// TIA Portal project "Projekt_v2" (V13)
// Vorlageprojekt für das Buch mit Zielsystem S7-1200

(* hardware
DEVICE "S7-1200-Station_1"  S7-1200 Station
   slot 0: "Baugruppenträger_0"  Rack  V1.0
   slot 1: "PLC_1"  CPU 1214C DC/DC/Rly  6ES7 214-1HG40-0XB0  V4.1
   slot 2: "DQ 16xRelay_1"  6ES7 222-1HH30-0XB0  V1.0
   slot 3: "DI 16x24VDC_1"  6ES7 221-1BH32-0XB0  V2.0
*)

// ===== PLC "PLC_1"  CPU 1214C DC/DC/Rly =====

VAR_GLOBAL   // PLC tag table "Standard-Variablentabelle"
   "Tag_2" AT %I0.0 : Bool;
   "Tag_3" AT %I0.1 : Bool;
   "Start btn" AT %I0.2 : Bool;
   "Emergency" AT %I0.4 : Bool;
   "Stop btn" AT %I0.3 : Bool;
   "Sstart" AT %I0.5 : Bool;
   "VS sorting 1" AT %ID38 : DWord;
   "VS sorting2" AT %ID34 : DWord;
   "ColorStopS" AT %I0.6 : Bool;
   "Threshold1" AT %I0.7 : Bool;
   "ResetBufor" AT %I1.0 : Bool;
   "ErrorSensor" AT %I1.1 : Bool;
   "SolveError" AT %I1.2 : Bool;
   "PallPalletAtEntry" AT %I2.0 : Bool;
   "PallPalletAtExit" AT %I2.1 : Bool;
   "PallPalletLoaded" AT %I2.2 : Bool;
   "PallBoxAtEntry" AT %I2.3 : Bool;
   "PallPusherLimit" AT %I2.4 : Bool;
   "PallPlateLimit" AT %I2.5 : Bool;
   "PallClamped" AT %I2.6 : Bool;
   "PallElevatorMoving" AT %I2.7 : Bool;
   "PallReset" AT %I1.3 : Bool;
   "Tag_1" AT %Q0.0 : Bool;
   "Start LED" AT %Q0.2 : Bool;
   "Stop LED" AT %Q0.3 : Bool;
   "ALARM" AT %Q0.4 : Bool;
   "1st Belt" AT %Q2.2 : Bool;
   "Sorter" AT %Q2.3 : Bool;
   "SorterToRight" AT %Q2.1 : Bool;
   "Arm4th" AT %Q0.7 : Bool;
   "Arm2nd" AT %Q1.0 : Bool;
   "2nd Belt" AT %Q2.4 : Bool;
   "3rd Arm" AT %Q1.1 : Bool;
   "PallPalletFeeder" AT %Q3.0 : Bool;
   "PallLoadPallet" AT %Q3.1 : Bool;
   "PallExitConveyor" AT %Q3.2 : Bool;
   "PallMoveToLimit" AT %Q3.3 : Bool;
   "PallElevatorUp" AT %Q3.4 : Bool;
   "PallElevatorDown" AT %Q3.5 : Bool;
   "PallBoxFeeder" AT %Q3.6 : Bool;
   "PallTurn" AT %Q3.7 : Bool;
   "PallPush" AT %Q4.0 : Bool;
   "PallLoadBelt" AT %Q4.1 : Bool;
   "PallClamp" AT %Q4.2 : Bool;
   "PallOpenPlate" AT %Q4.3 : Bool;
   "Priv ST" AT %M0.0 : Bool;
   "START" AT %M0.1 : Bool;
   "Tag_4" AT %M0.2 : Bool;
   "Tag_5" AT %M0.3 : Bool;
   "Tag_6" AT %M0.4 : Bool;
   "Change direction" AT %M0.5 : Bool;
   "Green Mark" AT %M1.0 : Bool;
   "BlueMark" AT %M1.1 : Bool;
   "BuforSort" AT %M8.0 : Bool;
   "FULLSORT" AT %M1.2 : Bool;
   "MetalMark" AT %M1.3 : Bool;
   "ERROR" AT %M8.2 : Bool;
   "ErrorMark" AT %M1.4 : Bool;
   "PallOpenPlateRising" AT %M3.0 : Bool;
   "PallPalletAtExitRising" AT %M3.1 : Bool;
   "PallElevatorPosition" AT %M3.2 : Bool;
   "PallBoxAtEntryRising" AT %M3.3 : Bool;
   "PallPusherLimitRising" AT %M3.4 : Bool;
   "PallPlateLimitRising" AT %M3.5 : Bool;
   "PallElevatorDownRising" AT %M3.6 : Bool;
   "PallBoxesRows" AT %MW10 : Int;
   "PallNumberBoxRows" AT %MW14 : Int;
   "PallAlturningFlag" AT %M3.7 : Bool;
   "PallPushRising" AT %M4.0 : Bool;
   "PallElevatorMovingFalling" AT %M4.1 : Bool;
   "PallPushBoxRising" AT %M4.2 : Bool;
   "PallPusherLimitFalling" AT %M4.3 : Bool;
   "PallElevatorDownRising2" AT %M4.4 : Bool;
   "SORTERisFULL" AT %M8.3 : Bool;
   "4th belt" AT %Q2.5 : Bool;
   "Arm 4th" AT %Q1.2 : Bool;
   "1st pivot" AT %Q1.3 : Bool;
   "2nd pivot" AT %Q1.4 : Bool;
   "3rd pivot" AT %Q1.5 : Bool;
   "4th pivot" AT %Q1.6 : Bool;
   "GreenTakeOFF" AT %Q0.5 : Bool;
   "BlueTakeOFF" AT %Q0.6 : Bool;
   "MetalTakeOFF" AT %Q1.7 : Bool;
   "ErrorTakeOFF" AT %Q2.0 : Bool;
END_VAR

VAR_GLOBAL CONSTANT   // PLC tag table "Standard-Variablentabelle"
   "Test" : Int := 3;
END_VAR

// folder: System blocks/Program resources

DATA_BLOCK "IEC_Timer_0_DB"   // DB1
{ S7_Optimized_Access := 'FALSE' }
AUTHOR : Simatic
FAMILY : IEC
NAME : IEC_TMR
VERSION : 1.0
// stored: InstanceOfName ?
"?"
BEGIN
END_DATA_BLOCK

DATA_BLOCK "IEC_Timer_0_DB_1"   // DB2
{ S7_Optimized_Access := 'FALSE' }
AUTHOR : Simatic
FAMILY : IEC
NAME : IEC_TMR
VERSION : 1.0
// stored: InstanceOfName ?
"?"
BEGIN
END_DATA_BLOCK

DATA_BLOCK "IEC_Timer_0_DB_2"   // DB3
{ S7_Optimized_Access := 'FALSE' }
AUTHOR : Simatic
FAMILY : IEC
NAME : IEC_TMR
VERSION : 1.0
// stored: InstanceOfName ?
"?"
BEGIN
END_DATA_BLOCK

DATA_BLOCK "IEC_Timer_0_DB_3"   // DB4
{ S7_Optimized_Access := 'FALSE' }
AUTHOR : Simatic
FAMILY : IEC
NAME : IEC_TMR
VERSION : 1.0
// stored: InstanceOfName ?
"?"
BEGIN
END_DATA_BLOCK

DATA_BLOCK "IEC_Timer_0_DB_4"   // DB5
{ S7_Optimized_Access := 'FALSE' }
AUTHOR : Simatic
FAMILY : IEC
NAME : IEC_TMR
VERSION : 1.0
// stored: InstanceOfName ?
"?"
BEGIN
END_DATA_BLOCK

DATA_BLOCK "IEC_Timer_0_DB_5"   // DB6
{ S7_Optimized_Access := 'FALSE' }
AUTHOR : Simatic
FAMILY : IEC
NAME : IEC_TMR
VERSION : 1.0
// stored: InstanceOfName ?
"?"
BEGIN
END_DATA_BLOCK

DATA_BLOCK "IEC_Timer_0_DB_6"   // DB7
{ S7_Optimized_Access := 'FALSE' }
AUTHOR : Simatic
FAMILY : IEC
NAME : IEC_TMR
VERSION : 1.0
// stored: InstanceOfName ?
"?"
BEGIN
END_DATA_BLOCK

DATA_BLOCK "Layer_Counter"   // DB8
{ S7_Optimized_Access := 'FALSE' }
AUTHOR : Simatic
FAMILY : IEC
NAME : CNTR
VERSION : 1.0
// stored: InstanceOfName ?
"?"
BEGIN
END_DATA_BLOCK

DATA_BLOCK "Off_Delay_Timer"   // DB10
{ S7_Optimized_Access := 'FALSE' }
AUTHOR : Simatic
FAMILY : IEC
NAME : IEC_TMR
VERSION : 1.0
// stored: InstanceOfName ?
"?"
BEGIN
END_DATA_BLOCK

DATA_BLOCK "Boxes_In_Row"   // DB11
{ S7_Optimized_Access := 'FALSE' }
AUTHOR : Simatic
FAMILY : IEC
NAME : CNTR
VERSION : 1.0
// stored: InstanceOfName ?
"?"
BEGIN
END_DATA_BLOCK

DATA_BLOCK "Number_of_Row"   // DB12
{ S7_Optimized_Access := 'FALSE' }
AUTHOR : Simatic
FAMILY : IEC
NAME : CNTR
VERSION : 1.0
// stored: InstanceOfName ?
"?"
BEGIN
END_DATA_BLOCK

DATA_BLOCK "Pall_Push_Timer"   // DB14
{ S7_Optimized_Access := 'FALSE' }
AUTHOR : Simatic
FAMILY : IEC
NAME : IEC_TMR
VERSION : 1.0
// stored: InstanceOfName ?
"?"
BEGIN
END_DATA_BLOCK

DATA_BLOCK "Pall_Open_Plate_Timer"   // DB15
{ S7_Optimized_Access := 'FALSE' }
AUTHOR : Simatic
FAMILY : IEC
NAME : IEC_TMR
VERSION : 1.0
// stored: InstanceOfName ?
"?"
BEGIN
END_DATA_BLOCK

// folder: (top level)

FUNCTION "Program" : Void   // FC1, LAD
{ S7_Optimized_Access := 'FALSE' }
VERSION : 0.1
   VAR_TEMP   // added for the SCL form of the ladder/FBD networks
      _w1 : Bool;
   END_VAR
BEGIN

REGION Network 1
   // Status: Start
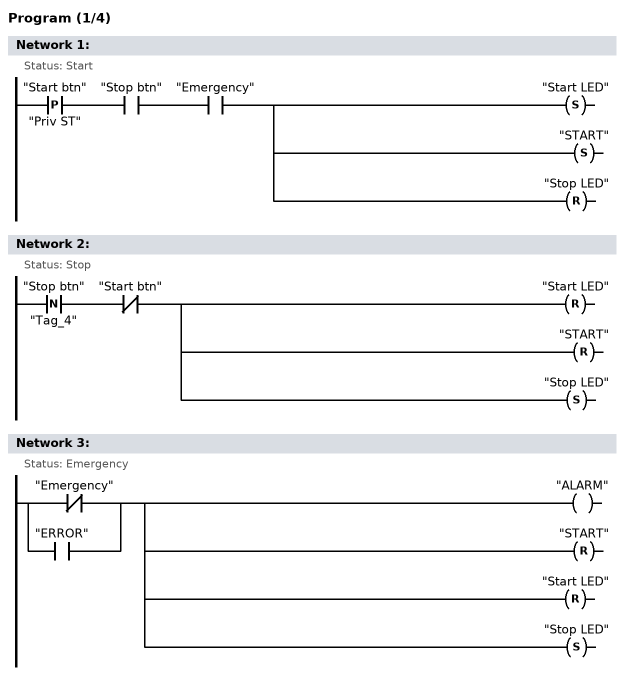
   RUNG wire#powerrail
      P_Contact(operand := "Start btn", bit := "Priv ST")
      Contact( "Stop btn" )
      Contact( "Emergency" )
      wire#w1
      S_Coil( "Start LED" )
   END_RUNG
   RUNG wire#w1
      S_Coil( "START" )
   END_RUNG
   RUNG wire#w1
      R_Coil( "Stop LED" )
   END_RUNG
   // the same network as SCL:
   #_w1 := "Start btn" AND NOT "Priv ST";   // rising edge of "Start btn"
   "Priv ST" := "Start btn";
   IF #_w1 AND "Stop btn" AND "Emergency" THEN
       "Start LED" := TRUE;
       "START" := TRUE;
       "Stop LED" := FALSE;
   END_IF;
END_REGION

REGION Network 2
   // Status: Stop
   RUNG wire#powerrail
      N_Contact(operand := "Stop btn", bit := "Tag_4")
      I_Contact( "Start btn" )
      wire#w1
      R_Coil( "Start LED" )
   END_RUNG
   RUNG wire#w1
      R_Coil( "START" )
   END_RUNG
   RUNG wire#w1
      S_Coil( "Stop LED" )
   END_RUNG
   // the same network as SCL:
   #_w1 := NOT "Stop btn" AND "Tag_4";   // falling edge of "Stop btn"
   "Tag_4" := "Stop btn";
   IF #_w1 AND NOT "Start btn" THEN
       "Start LED" := FALSE;
       "START" := FALSE;
       "Stop LED" := TRUE;
   END_IF;
END_REGION

REGION Network 3
   // Status: Emergency
   RUNG wire#powerrail
      I_Contact( "Emergency" )
      wire#w1
      Coil( "ALARM" )
   END_RUNG
   RUNG wire#powerrail
      Contact( "ERROR" )
   END_RUNG wire#w1
   RUNG wire#w1
      R_Coil( "START" )
   END_RUNG
   RUNG wire#w1
      R_Coil( "Start LED" )
   END_RUNG
   RUNG wire#w1
      S_Coil( "Stop LED" )
   END_RUNG
   // the same network as SCL:
   "ALARM" := NOT "Emergency" OR "ERROR";
   IF "ALARM" THEN
       "START" := FALSE;
       "Start LED" := FALSE;
       "Stop LED" := TRUE;
   END_IF;
END_REGION

REGION Network 4
   // 1st settings
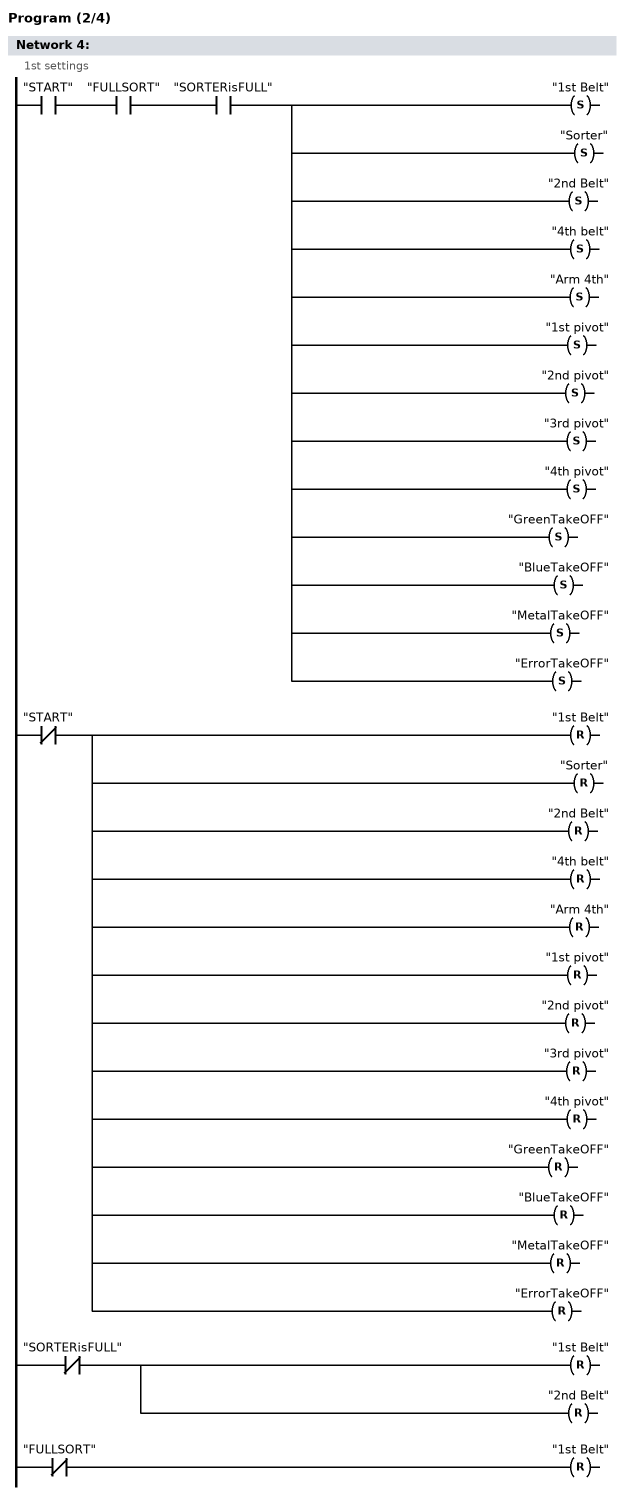
   RUNG wire#powerrail
      Contact( "START" )
      Contact( "FULLSORT" )
      Contact( "SORTERisFULL" )
      wire#w1
      S_Coil( "1st Belt" )
   END_RUNG
   RUNG wire#w1
      S_Coil( "Sorter" )
   END_RUNG
   RUNG wire#w1
      S_Coil( "2nd Belt" )
   END_RUNG
   RUNG wire#w1
      S_Coil( "4th belt" )
   END_RUNG
   RUNG wire#w1
      S_Coil( "Arm 4th" )
   END_RUNG
   RUNG wire#w1
      S_Coil( "1st pivot" )
   END_RUNG
   RUNG wire#w1
      S_Coil( "2nd pivot" )
   END_RUNG
   RUNG wire#w1
      S_Coil( "3rd pivot" )
   END_RUNG
   RUNG wire#w1
      S_Coil( "4th pivot" )
   END_RUNG
   RUNG wire#w1
      S_Coil( "GreenTakeOFF" )
   END_RUNG
   RUNG wire#w1
      S_Coil( "BlueTakeOFF" )
   END_RUNG
   RUNG wire#w1
      S_Coil( "MetalTakeOFF" )
   END_RUNG
   RUNG wire#w1
      S_Coil( "ErrorTakeOFF" )
   END_RUNG
   RUNG wire#powerrail
      I_Contact( "START" )
      wire#w2
      R_Coil( "1st Belt" )
   END_RUNG
   RUNG wire#w2
      R_Coil( "Sorter" )
   END_RUNG
   RUNG wire#w2
      R_Coil( "2nd Belt" )
   END_RUNG
   RUNG wire#w2
      R_Coil( "4th belt" )
   END_RUNG
   RUNG wire#w2
      R_Coil( "Arm 4th" )
   END_RUNG
   RUNG wire#w2
      R_Coil( "1st pivot" )
   END_RUNG
   RUNG wire#w2
      R_Coil( "2nd pivot" )
   END_RUNG
   RUNG wire#w2
      R_Coil( "3rd pivot" )
   END_RUNG
   RUNG wire#w2
      R_Coil( "4th pivot" )
   END_RUNG
   RUNG wire#w2
      R_Coil( "GreenTakeOFF" )
   END_RUNG
   RUNG wire#w2
      R_Coil( "BlueTakeOFF" )
   END_RUNG
   RUNG wire#w2
      R_Coil( "MetalTakeOFF" )
   END_RUNG
   RUNG wire#w2
      R_Coil( "ErrorTakeOFF" )
   END_RUNG
   RUNG wire#powerrail
      I_Contact( "SORTERisFULL" )
      wire#w3
      R_Coil( "1st Belt" )
   END_RUNG
   RUNG wire#w3
      R_Coil( "2nd Belt" )
   END_RUNG
   RUNG wire#powerrail
      I_Contact( "FULLSORT" )
      R_Coil( "1st Belt" )
   END_RUNG
   // the same network as SCL:
   IF "START" AND "FULLSORT" AND "SORTERisFULL" THEN
       "1st Belt" := TRUE;
       "Sorter" := TRUE;
       "2nd Belt" := TRUE;
       "4th belt" := TRUE;
       "Arm 4th" := TRUE;
       "1st pivot" := TRUE;
       "2nd pivot" := TRUE;
       "3rd pivot" := TRUE;
       "4th pivot" := TRUE;
       "GreenTakeOFF" := TRUE;
       "BlueTakeOFF" := TRUE;
       "MetalTakeOFF" := TRUE;
       "ErrorTakeOFF" := TRUE;
   END_IF;
   IF NOT "START" THEN
       "1st Belt" := FALSE;
       "Sorter" := FALSE;
       "2nd Belt" := FALSE;
       "4th belt" := FALSE;
       "Arm 4th" := FALSE;
       "1st pivot" := FALSE;
       "2nd pivot" := FALSE;
       "3rd pivot" := FALSE;
       "4th pivot" := FALSE;
       "GreenTakeOFF" := FALSE;
       "BlueTakeOFF" := FALSE;
       "MetalTakeOFF" := FALSE;
       "ErrorTakeOFF" := FALSE;
   END_IF;
   IF NOT "SORTERisFULL" THEN
       "1st Belt" := FALSE;
       "2nd Belt" := FALSE;
   END_IF;
   IF NOT "FULLSORT" THEN "1st Belt" := FALSE; END_IF;
END_REGION

REGION Network 5
   // 1st sorting boxes vs color things
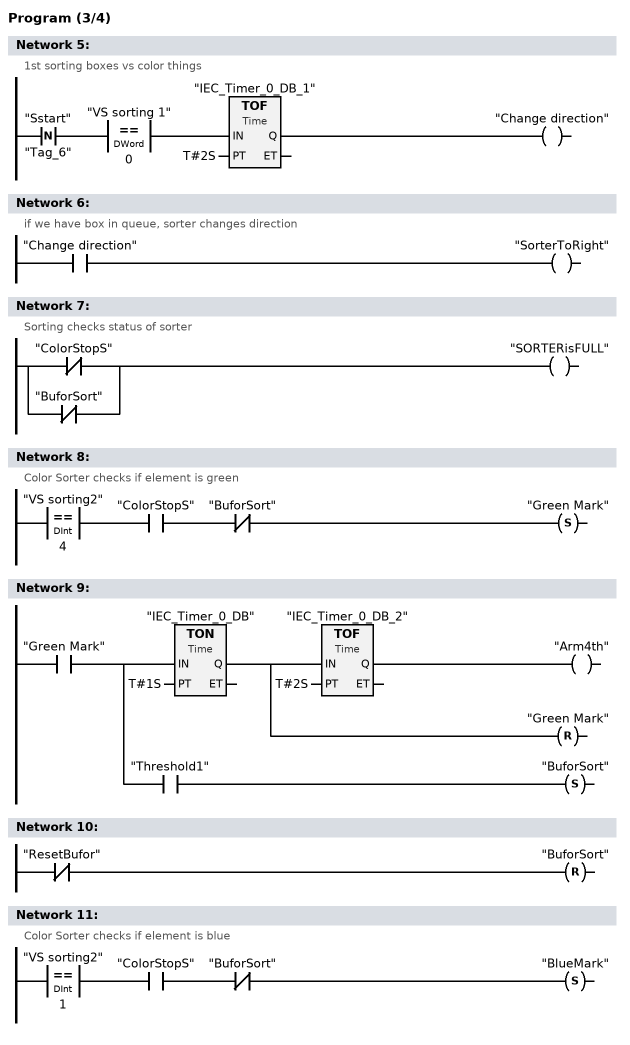
   #_w1 := NOT "Sstart" AND "Tag_6";   // falling edge of "Sstart"
   "Tag_6" := "Sstart";
   "IEC_Timer_0_DB_1".TOF(IN := #_w1 AND ("VS sorting 1" = 0), PT := T#2S);
   "Change direction" := "IEC_Timer_0_DB_1".Q;
END_REGION

REGION Network 6
   // if we have box in queue, sorter changes direction
   RUNG wire#powerrail
      Contact( "Change direction" )
      Coil( "SorterToRight" )
   END_RUNG
   // the same network as SCL:
   "SorterToRight" := "Change direction";
END_REGION

REGION Network 7
   // Sorting checks status of sorter
   RUNG wire#powerrail
      I_Contact( "ColorStopS" )
      wire#w1
      Coil( "SORTERisFULL" )
   END_RUNG
   RUNG wire#powerrail
      I_Contact( "BuforSort" )
   END_RUNG wire#w1
   // the same network as SCL:
   "SORTERisFULL" := NOT "ColorStopS" OR NOT "BuforSort";
END_REGION

REGION Network 8
   // Color Sorter checks if element is green
   RUNG wire#powerrail
      { S7_Templates := "SrcType := DInt" } EQ_Contact(in1 := "VS sorting2", in2 := 4)
      Contact( "ColorStopS" )
      I_Contact( "BuforSort" )
      S_Coil( "Green Mark" )
   END_RUNG
   // the same network as SCL:
   IF ("VS sorting2" = 4) AND "ColorStopS" AND NOT "BuforSort" THEN "Green Mark" := TRUE; END_IF;
END_REGION

REGION Network 9
   "IEC_Timer_0_DB".TON(IN := "Green Mark", PT := T#1S);
   "IEC_Timer_0_DB_2".TOF(IN := "IEC_Timer_0_DB".Q, PT := T#2S);
   "Arm4th" := "IEC_Timer_0_DB_2".Q;
   #_w1 := "Green Mark";
   IF "IEC_Timer_0_DB".Q THEN "Green Mark" := FALSE; END_IF;
   IF #_w1 AND "Threshold1" THEN "BuforSort" := TRUE; END_IF;
END_REGION

REGION Network 10
   RUNG wire#powerrail
      I_Contact( "ResetBufor" )
      R_Coil( "BuforSort" )
   END_RUNG
   // the same network as SCL:
   IF NOT "ResetBufor" THEN "BuforSort" := FALSE; END_IF;
END_REGION

REGION Network 11
   // Color Sorter checks if element is blue
   RUNG wire#powerrail
      { S7_Templates := "SrcType := DInt" } EQ_Contact(in1 := "VS sorting2", in2 := 1)
      Contact( "ColorStopS" )
      I_Contact( "BuforSort" )
      S_Coil( "BlueMark" )
   END_RUNG
   // the same network as SCL:
   IF ("VS sorting2" = 1) AND "ColorStopS" AND NOT "BuforSort" THEN "BlueMark" := TRUE; END_IF;
END_REGION

REGION Network 12
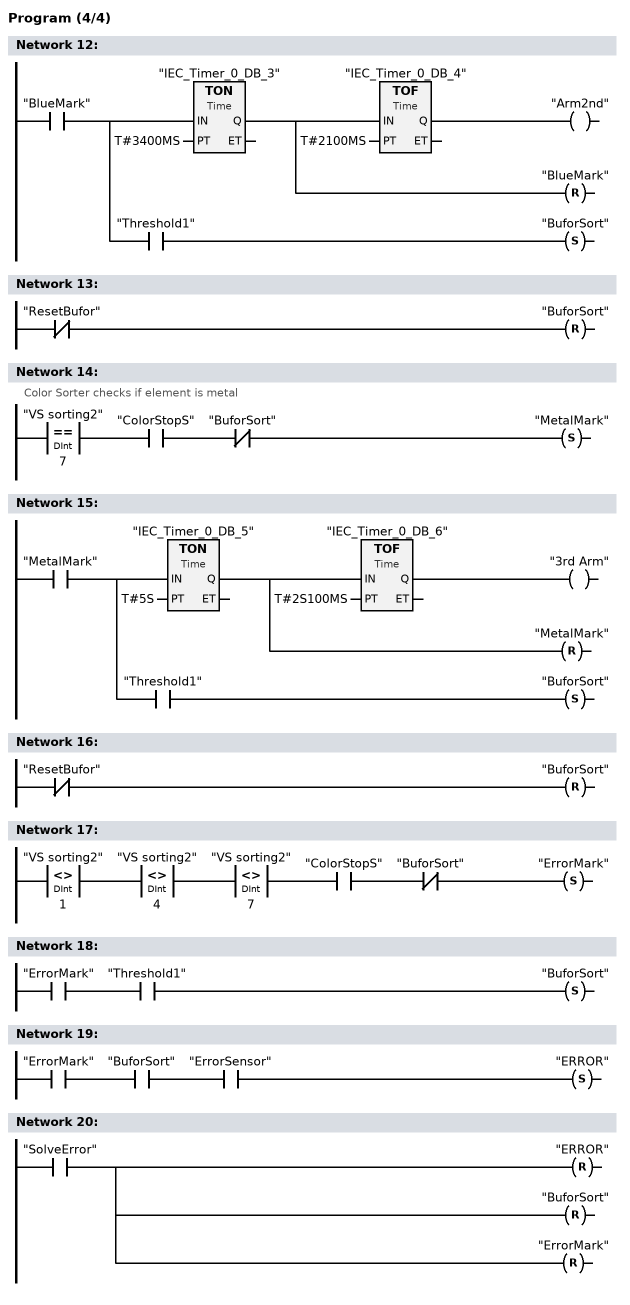
   "IEC_Timer_0_DB_3".TON(IN := "BlueMark", PT := T#3400MS);
   "IEC_Timer_0_DB_4".TOF(IN := "IEC_Timer_0_DB_3".Q, PT := T#2100MS);
   "Arm2nd" := "IEC_Timer_0_DB_4".Q;
   #_w1 := "BlueMark";
   IF "IEC_Timer_0_DB_3".Q THEN "BlueMark" := FALSE; END_IF;
   IF #_w1 AND "Threshold1" THEN "BuforSort" := TRUE; END_IF;
END_REGION

REGION Network 13
   RUNG wire#powerrail
      I_Contact( "ResetBufor" )
      R_Coil( "BuforSort" )
   END_RUNG
   // the same network as SCL:
   IF NOT "ResetBufor" THEN "BuforSort" := FALSE; END_IF;
END_REGION

REGION Network 14
   // Color Sorter checks if element is metal
   RUNG wire#powerrail
      { S7_Templates := "SrcType := DInt" } EQ_Contact(in1 := "VS sorting2", in2 := 7)
      Contact( "ColorStopS" )
      I_Contact( "BuforSort" )
      S_Coil( "MetalMark" )
   END_RUNG
   // the same network as SCL:
   IF ("VS sorting2" = 7) AND "ColorStopS" AND NOT "BuforSort" THEN "MetalMark" := TRUE; END_IF;
END_REGION

REGION Network 15
   "IEC_Timer_0_DB_5".TON(IN := "MetalMark", PT := T#5S);
   "IEC_Timer_0_DB_6".TOF(IN := "IEC_Timer_0_DB_5".Q, PT := T#2S100MS);
   "3rd Arm" := "IEC_Timer_0_DB_6".Q;
   #_w1 := "MetalMark";
   IF "IEC_Timer_0_DB_5".Q THEN "MetalMark" := FALSE; END_IF;
   IF #_w1 AND "Threshold1" THEN "BuforSort" := TRUE; END_IF;
END_REGION

REGION Network 16
   RUNG wire#powerrail
      I_Contact( "ResetBufor" )
      R_Coil( "BuforSort" )
   END_RUNG
   // the same network as SCL:
   IF NOT "ResetBufor" THEN "BuforSort" := FALSE; END_IF;
END_REGION

REGION Network 17
   RUNG wire#powerrail
      { S7_Templates := "SrcType := DInt" } NE_Contact(in1 := "VS sorting2", in2 := 1)
      { S7_Templates := "SrcType := DInt" } NE_Contact(in1 := "VS sorting2", in2 := 4)
      { S7_Templates := "SrcType := DInt" } NE_Contact(in1 := "VS sorting2", in2 := 7)
      Contact( "ColorStopS" )
      I_Contact( "BuforSort" )
      S_Coil( "ErrorMark" )
   END_RUNG
   // the same network as SCL:
   IF ("VS sorting2" <> 1) AND ("VS sorting2" <> 4) AND ("VS sorting2" <> 7) AND "ColorStopS" AND NOT "BuforSort" THEN
       "ErrorMark" := TRUE;
   END_IF;
END_REGION

REGION Network 18
   RUNG wire#powerrail
      Contact( "ErrorMark" )
      Contact( "Threshold1" )
      S_Coil( "BuforSort" )
   END_RUNG
   // the same network as SCL:
   IF "ErrorMark" AND "Threshold1" THEN "BuforSort" := TRUE; END_IF;
END_REGION

REGION Network 19
   RUNG wire#powerrail
      Contact( "ErrorMark" )
      Contact( "BuforSort" )
      Contact( "ErrorSensor" )
      S_Coil( "ERROR" )
   END_RUNG
   // the same network as SCL:
   IF "ErrorMark" AND "BuforSort" AND "ErrorSensor" THEN "ERROR" := TRUE; END_IF;
END_REGION

REGION Network 20
   RUNG wire#powerrail
      Contact( "SolveError" )
      wire#w1
      R_Coil( "ERROR" )
   END_RUNG
   RUNG wire#w1
      R_Coil( "BuforSort" )
   END_RUNG
   RUNG wire#w1
      R_Coil( "ErrorMark" )
   END_RUNG
   // the same network as SCL:
   IF "SolveError" THEN
       "ERROR" := FALSE;
       "BuforSort" := FALSE;
       "ErrorMark" := FALSE;
   END_IF;
END_REGION
END_FUNCTION

FUNCTION "Palletizer" : Void   // FC2, LAD
{ S7_Optimized_Access := 'FALSE' }
VERSION : 0.1
   VAR_TEMP   // added for the SCL form of the ladder/FBD networks
      _w1 : Bool;
      _w2 : Bool;
      _w3 : Bool;
      _w4 : Bool;
      _w5 : Bool;
      _w6 : Bool;
      _w7 : Bool;
      _w8 : Bool;
      _w9 : Bool;
      _w10 : Bool;
      _w11 : Bool;
   END_VAR
BEGIN

REGION Network 1: Loading / Unloading Pallets
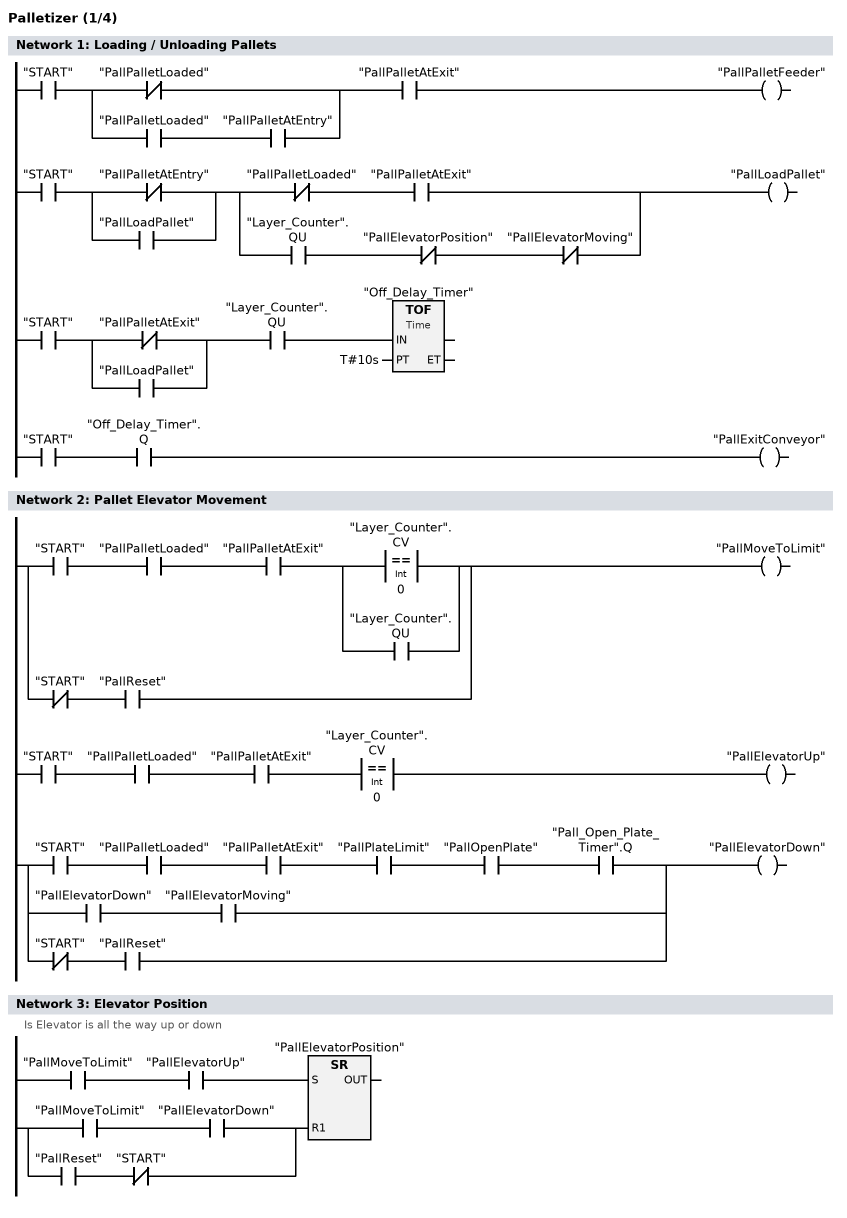
   "PallPalletFeeder" := "START" AND (NOT "PallPalletLoaded" OR ("PallPalletLoaded" AND "PallPalletAtEntry")) AND "PallPalletAtExit";
   "PallLoadPallet" := "START" AND (NOT "PallPalletAtEntry" OR "PallLoadPallet") AND ((NOT "PallPalletLoaded" AND "PallPalletAtExit") OR ("Layer_Counter".QU AND NOT "PallElevatorPosition" AND NOT "PallElevatorMoving"));
   "Off_Delay_Timer".TOF(IN := "START" AND (NOT "PallPalletAtExit" OR "PallLoadPallet") AND "Layer_Counter".QU,
                         PT := T#10s);
   "PallExitConveyor" := "START" AND "Off_Delay_Timer".Q;
END_REGION

REGION Network 2: Pallet Elevator Movement
   RUNG wire#powerrail
      Contact( "START" )
      Contact( "PallPalletLoaded" )
      Contact( "PallPalletAtExit" )
      wire#w1
      { S7_Templates := "SrcType := Int" } EQ_Contact(in1 := "Layer_Counter".CV, in2 := 0)
      wire#w2
      Coil( "PallMoveToLimit" )
   END_RUNG
   RUNG wire#w1
      Contact( "Layer_Counter".QU )
   END_RUNG wire#w2
   RUNG wire#powerrail
      I_Contact( "START" )
      Contact( "PallReset" )
   END_RUNG wire#w2
   RUNG wire#powerrail
      Contact( "START" )
      Contact( "PallPalletLoaded" )
      Contact( "PallPalletAtExit" )
      { S7_Templates := "SrcType := Int" } EQ_Contact(in1 := "Layer_Counter".CV, in2 := 0)
      Coil( "PallElevatorUp" )
   END_RUNG
   RUNG wire#powerrail
      Contact( "START" )
      Contact( "PallPalletLoaded" )
      Contact( "PallPalletAtExit" )
      Contact( "PallPlateLimit" )
      Contact( "PallOpenPlate" )
      Contact( "Pall_Open_Plate_Timer".Q )
      wire#w3
      Coil( "PallElevatorDown" )
   END_RUNG
   RUNG wire#powerrail
      Contact( "PallElevatorDown" )
      Contact( "PallElevatorMoving" )
   END_RUNG wire#w3
   RUNG wire#powerrail
      I_Contact( "START" )
      Contact( "PallReset" )
   END_RUNG wire#w3
   // the same network as SCL:
   "PallMoveToLimit" := ("START" AND "PallPalletLoaded" AND "PallPalletAtExit" AND (("Layer_Counter".CV = 0) OR "Layer_Counter".QU)) OR (NOT "START" AND "PallReset");
   "PallElevatorUp" := "START" AND "PallPalletLoaded" AND "PallPalletAtExit" AND ("Layer_Counter".CV = 0);
   "PallElevatorDown" := ("START" AND "PallPalletLoaded" AND "PallPalletAtExit" AND "PallPlateLimit" AND "PallOpenPlate" AND "Pall_Open_Plate_Timer".Q) OR ("PallElevatorDown" AND "PallElevatorMoving") OR (NOT "START" AND "PallReset");
END_REGION

REGION Network 3: Elevator Position
   // Is Elevator is all the way up or down
   RUNG wire#powerrail
      Contact( "PallMoveToLimit" )
      Contact( "PallElevatorUp" )
      S_SR(operand := "PallElevatorPosition", r1 := wire#w1)
   END_RUNG
   RUNG wire#powerrail
      Contact( "PallMoveToLimit" )
      Contact( "PallElevatorDown" )
   END_RUNG wire#w1
   RUNG wire#powerrail
      Contact( "PallReset" )
      I_Contact( "START" )
   END_RUNG wire#w1
   // the same network as SCL:
   IF "PallMoveToLimit" AND "PallElevatorUp" THEN
       "PallElevatorPosition" := TRUE;   // SR flip-flop
   END_IF;
   IF ("PallMoveToLimit" AND "PallElevatorDown") OR ("PallReset" AND NOT "START") THEN
       "PallElevatorPosition" := FALSE;
   END_IF;
END_REGION

REGION Network 4: Number of Layers on the Pallet
   // Couter tracks how many layers are on pallet
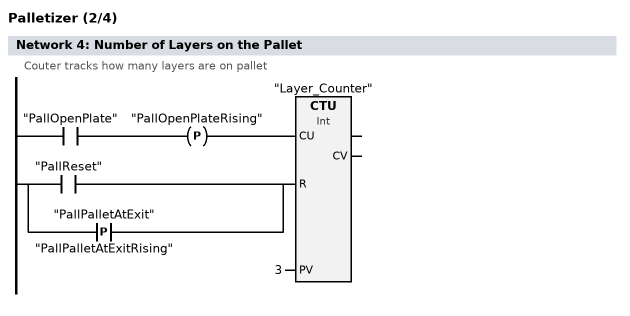
   #_w1 := "PallOpenPlate" AND NOT "PallOpenPlateRising";   // rising edge
   "PallOpenPlateRising" := "PallOpenPlate";
   #_w2 := "PallPalletAtExit" AND NOT "PallPalletAtExitRising";   // rising edge of "PallPalletAtExit"
   "PallPalletAtExitRising" := "PallPalletAtExit";
   "Layer_Counter".CTU(CU := #_w1, R := "PallReset" OR #_w2, PV := 3);
END_REGION

REGION Network 5: Boxes on Layers
   // 6 boxes on layer. Each Layer is alturnating
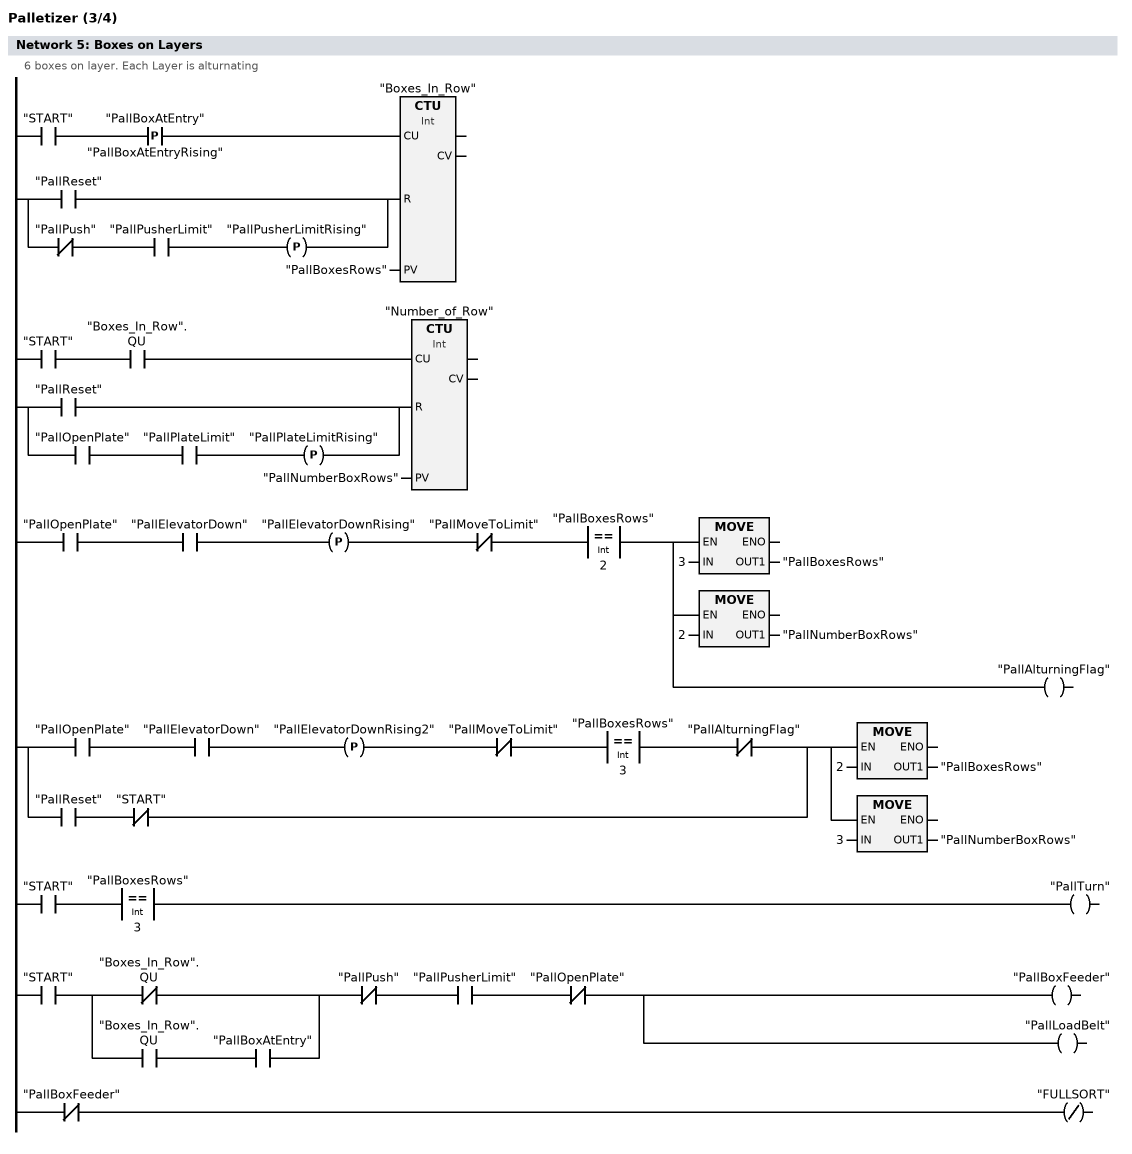
   #_w1 := "START" AND "PallBoxAtEntry" AND NOT "PallBoxAtEntryRising";   // rising edge of "PallBoxAtEntry"
   "PallBoxAtEntryRising" := "PallBoxAtEntry";
   #_w2 := NOT "PallPush" AND "PallPusherLimit";
   #_w3 := #_w2 AND NOT "PallPusherLimitRising";   // rising edge
   "PallPusherLimitRising" := #_w2;
   "Boxes_In_Row".CTU(CU := #_w1, R := "PallReset" OR #_w3, PV := "PallBoxesRows");
   #_w4 := "PallOpenPlate" AND "PallPlateLimit";
   #_w5 := #_w4 AND NOT "PallPlateLimitRising";   // rising edge
   "PallPlateLimitRising" := #_w4;
   "Number_of_Row".CTU(CU := "START" AND "Boxes_In_Row".QU, R := "PallReset" OR #_w5, PV := "PallNumberBoxRows");
   #_w6 := "PallOpenPlate" AND "PallElevatorDown";
   #_w7 := #_w6 AND NOT "PallElevatorDownRising";   // rising edge
   "PallElevatorDownRising" := #_w6;
   #_w8 := #_w7 AND NOT "PallMoveToLimit" AND ("PallBoxesRows" = 2);
   IF #_w8 THEN
       "PallBoxesRows" := 3;
       "PallNumberBoxRows" := 2;
   END_IF;
   "PallAlturningFlag" := #_w8;
   #_w9 := "PallOpenPlate" AND "PallElevatorDown";
   #_w10 := #_w9 AND NOT "PallElevatorDownRising2";   // rising edge
   "PallElevatorDownRising2" := #_w9;
   #_w11 := (#_w10 AND NOT "PallMoveToLimit" AND ("PallBoxesRows" = 3) AND NOT "PallAlturningFlag") OR ("PallReset" AND NOT "START");
   IF #_w11 THEN
       "PallBoxesRows" := 2;
       "PallNumberBoxRows" := 3;
   END_IF;
   "PallTurn" := "START" AND ("PallBoxesRows" = 3);
   "PallBoxFeeder" := "START" AND (NOT "Boxes_In_Row".QU OR ("Boxes_In_Row".QU AND "PallBoxAtEntry")) AND NOT "PallPush" AND "PallPusherLimit" AND NOT "PallOpenPlate";
   "PallLoadBelt" := "PallBoxFeeder";
   "FULLSORT" := NOT (NOT "PallBoxFeeder");
END_REGION

REGION Network 6: Box Pusher
   // The pusher will push the boxes in the row onto the plate.
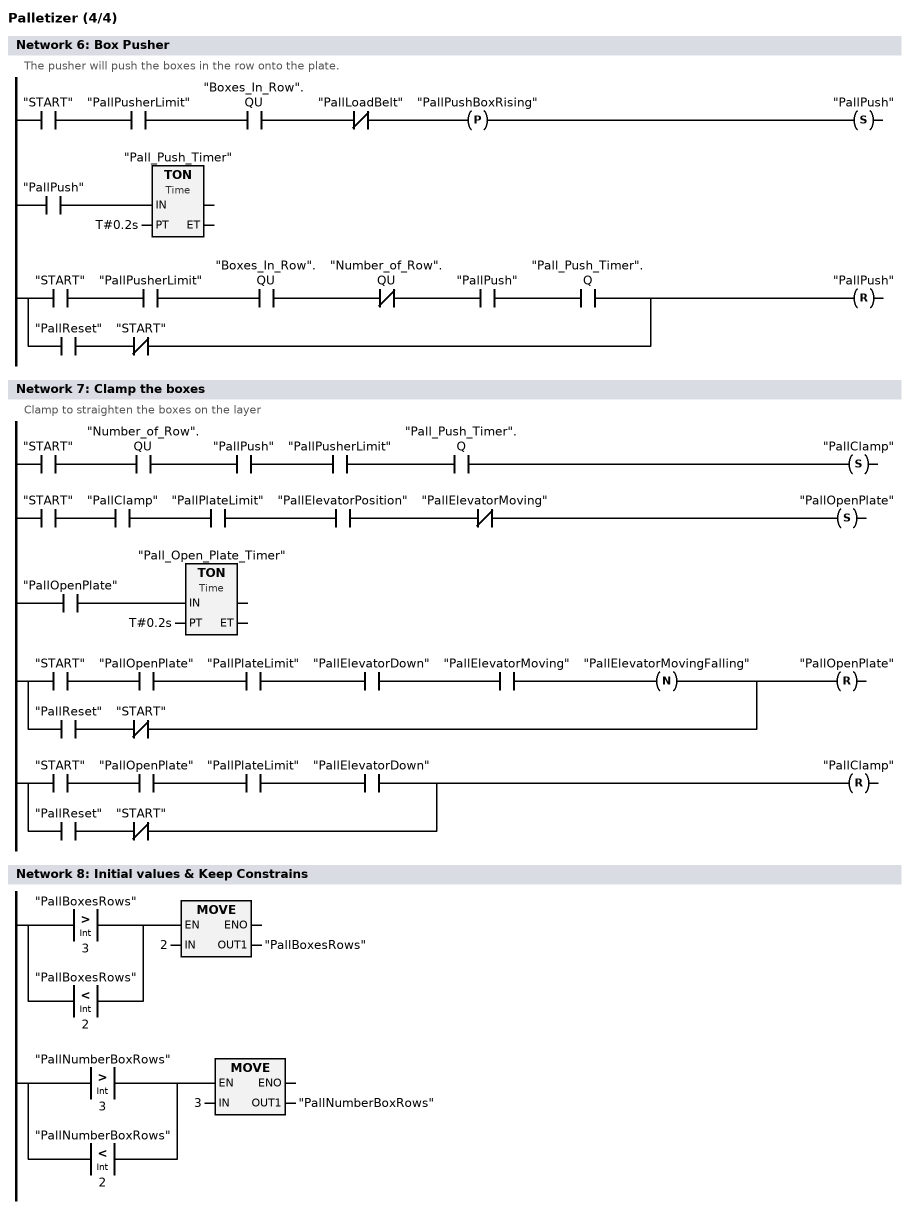
   #_w1 := "START" AND "PallPusherLimit" AND "Boxes_In_Row".QU AND NOT "PallLoadBelt";
   #_w2 := #_w1 AND NOT "PallPushBoxRising";   // rising edge
   "PallPushBoxRising" := #_w1;
   IF #_w2 THEN "PallPush" := TRUE; END_IF;
   "Pall_Push_Timer".TON(IN := "PallPush", PT := T#0.2s);
   IF ("START" AND "PallPusherLimit" AND "Boxes_In_Row".QU AND NOT "Number_of_Row".QU AND "PallPush" AND "Pall_Push_Timer".Q) OR ("PallReset" AND NOT "START") THEN
       "PallPush" := FALSE;
   END_IF;
END_REGION

REGION Network 7: Clamp the boxes
   // Clamp to straighten the boxes on the layer
   IF "START" AND "Number_of_Row".QU AND "PallPush" AND "PallPusherLimit" AND "Pall_Push_Timer".Q THEN
       "PallClamp" := TRUE;
   END_IF;
   IF "START" AND "PallClamp" AND "PallPlateLimit" AND "PallElevatorPosition" AND NOT "PallElevatorMoving" THEN
       "PallOpenPlate" := TRUE;
   END_IF;
   "Pall_Open_Plate_Timer".TON(IN := "PallOpenPlate", PT := T#0.2s);
   #_w1 := "START" AND "PallOpenPlate" AND "PallPlateLimit" AND "PallElevatorDown" AND "PallElevatorMoving";
   #_w2 := NOT #_w1 AND "PallElevatorMovingFalling";   // falling edge
   "PallElevatorMovingFalling" := #_w1;
   IF #_w2 OR ("PallReset" AND NOT "START") THEN "PallOpenPlate" := FALSE; END_IF;
   IF ("START" AND "PallOpenPlate" AND "PallPlateLimit" AND "PallElevatorDown") OR ("PallReset" AND NOT "START") THEN
       "PallClamp" := FALSE;
   END_IF;
END_REGION

REGION Network 8: Initial values & Keep Constrains
   RUNG wire#powerrail
      { S7_Templates := "SrcType := Int" } GT_Contact(in1 := "PallBoxesRows", in2 := 3)
      wire#w1
      Move(in := 2, out1 => "PallBoxesRows")
   END_RUNG
   RUNG wire#powerrail
      { S7_Templates := "SrcType := Int" } LT_Contact(in1 := "PallBoxesRows", in2 := 2)
   END_RUNG wire#w1
   RUNG wire#powerrail
      { S7_Templates := "SrcType := Int" } GT_Contact(in1 := "PallNumberBoxRows", in2 := 3)
      wire#w2
      Move(in := 3, out1 => "PallNumberBoxRows")
   END_RUNG
   RUNG wire#powerrail
      { S7_Templates := "SrcType := Int" } LT_Contact(in1 := "PallNumberBoxRows", in2 := 2)
   END_RUNG wire#w2
   // the same network as SCL:
   IF ("PallBoxesRows" > 3) OR ("PallBoxesRows" < 2) THEN "PallBoxesRows" := 2; END_IF;
   IF ("PallNumberBoxRows" > 3) OR ("PallNumberBoxRows" < 2) THEN "PallNumberBoxRows" := 3; END_IF;
END_REGION
END_FUNCTION

FUNCTION "MHJ-PLC-Lab-Function-S71200" : Void   // FC9000, SCL
{ S7_Optimized_Access := 'FALSE' }
VERSION : 0.1
BEGIN

   #Value:=PEEK(area := 16#82,
        dbNumber := 0,
        byteOffset := 511);
   #Value := #Value + 1;

   POKE(area := 16#82,
        dbNumber := 0,
        byteOffset := 511,
        value := #Value);

   POKE(area:=16#81,
        dbNumber:=0,
        byteOffset:=1016,
        value:=#Value_01_DW);
   POKE(area := 16#81,
        dbNumber := 0,
        byteOffset := 1020,
        value := #Value_02_DW);

   POKE(area := 16#81,
        dbNumber := 0,
        byteOffset := 511,
        value := B#16#00);

   FOR #forVal := 0 TO 120 DO
       FOR #forVal_2:=0 TO 10 DO
           #rdTimeReturn:=RD_SYS_T(#outputTime);
           #rdTimeReturn := WR_SYS_T(#outputTime);
           #rdTimeReturn := RD_SYS_T(#outputTime);
           #rdTimeReturn := WR_SYS_T(#outputTime);
       END_FOR;
       #SyncVal:= PEEK(area := 16#81,
                      dbNumber := 0,
                      byteOffset := 511);
       IF #SyncVal = #CompVal THEN
          GOTO M_1;
       END_IF;
   END_FOR;
   RETURN;

   M_1:
   POKE(area := 16#81,
        dbNumber := 0,
        byteOffset := 511,
        value := B#16#0);
END_FUNCTION

ORGANIZATION_BLOCK "Main"   // OB1, FBD, ProgramCycle
TITLE = "Main Program Sweep (Cycle)"
{ S7_Optimized_Access := 'FALSE' }
VERSION : 0.1
BEGIN

REGION Network 1
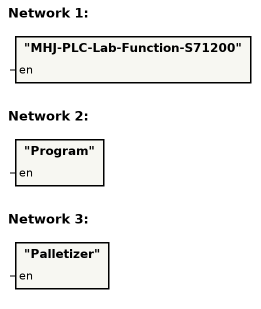
   "MHJ-PLC-Lab-Function-S71200"();
END_REGION

REGION Network 2
   "Program"();
END_REGION

REGION Network 3
   "Palletizer"();
END_REGION
END_ORGANIZATION_BLOCK